# EPICS autosave request: iocBoot/ioc13idd_linux/Galil_positions.req
file "CARS_56_motor_positions.req",      P=$(P)
file "CARS_8_motor_positions_sub.req",   P=$(P), M1=m65, M2=m66, M3=m67, M4=m68, M5=m69, M6=m70, M7=m71, M8=m72
file "CARS_8_motor_positions_sub.req",   P=$(P), M1=m73, M2=m74, M3=m75, M4=m76, M5=m77, M6=m78, M7=m79, M8=m80
